// TIA Portal V19 export
TYPE "ProjectInfo"
// stored: Access Published
   STRUCT
      Job : String[20];
      Revision : String[10];
      RevisionDate : DTL;
      Programmer : String[20];
      F_Signature : DWord;
      F_CompilationDate : DTL;
   END_STRUCT;
END_TYPE
